# EPICS autosave request: SIS8300App/Db/SIS8300_settings.req
$(P)$(R)NumTimePoints
$(P)$(R)TimeStep
$(P)$(R)AcquireTime
$(P)$(R)ClockSource
$(P)$(R)ClockFreq
$(P)$(R)ClockDiv
$(P)$(R)TrigSource
$(P)$(R)TrigDelay
$(P)$(R)TrigRepeat
$(P)$(R)RTMType

file "NDArrayBase_settings.req", P=$(P), R=$(R)
